// TIA Portal V20 export
DATA_BLOCK "IDB_Merging"   // DB27
// stored: InstanceOfName ProductionLine.FB_Merging, InstanceOfType FB, Namespace ProductionLine
"ProductionLine.FB_Merging"
   // VAR
   //    "Merge_A1.7.3" : "Global.FB_Merging";
   //    "Merge_A1.9.3" : "Global.FB_Merging";
   //    "Merge_B1.6.1" { S7_SetPoint := 'True'} : "Global.FB_Merging";
   // END_VAR
BEGIN
END_DATA_BLOCK
